Fanuc KAREL source: kc00004.KL

-- PROVISIONAL review KL for V770-1; original PC SHA256 3f642fc1f60d9fa99bafe436d7eb681e61b9652a297ab1aa3747f96ff87b73a7
-- Incomplete behavior may be omitted. Consult companion uncertainty JSON. Do not deploy.
PROGRAM KC00004
%NOLOCKGROUP
BEGIN
  -- UNRESOLVED_PC offsets 5-35; opcodes 27,22,22,22,2A,22,31
  -- UNRESOLVED_PC offsets 40-44; opcodes 7F
END KC00004
